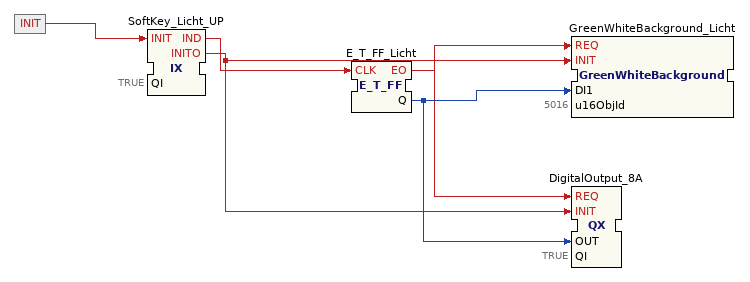
      FBS
        E_T_FF_Licht : E_T_FF;
        GreenWhiteBackground_Licht : GreenWhiteBackground(u16ObjId := 5016);
        DigitalOutput_8A : QX(QI := TRUE);
        SoftKey_Licht_UP : IX(QI := TRUE);
      END_FBS
      EVENT_CONNECTIONS
        SoftKey_Licht_UP.IND TO E_T_FF_Licht.CLK;
        E_T_FF_Licht.EO TO DigitalOutput_8A.REQ;
        E_T_FF_Licht.EO TO GreenWhiteBackground_Licht.REQ;
        SoftKey_Licht_UP.INITO TO GreenWhiteBackground_Licht.INIT;
        SoftKey_Licht_UP.INITO TO DigitalOutput_8A.INIT;
        INIT TO SoftKey_Licht_UP.INIT;
      END_CONNECTIONS
      DATA_CONNECTIONS
        E_T_FF_Licht.Q TO DigitalOutput_8A.OUT;
        E_T_FF_Licht.Q TO GreenWhiteBackground_Licht.DI1;
      END_CONNECTIONS
    END_SUBAPPLICATION
  END_APPLICATION
  APPLICATION Abscheider
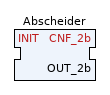
    SUBAPPLICATION Abscheider (* Abscheider *)
      EVENT_INPUT
        INIT; (* Service Initialization *)
      END_EVENT
      EVENT_OUTPUT
        CNF_2b; (* Execution Confirmation *)
      END_EVENT
      VAR_OUTPUT
        OUT_2b : BOOL;
      END_VAR
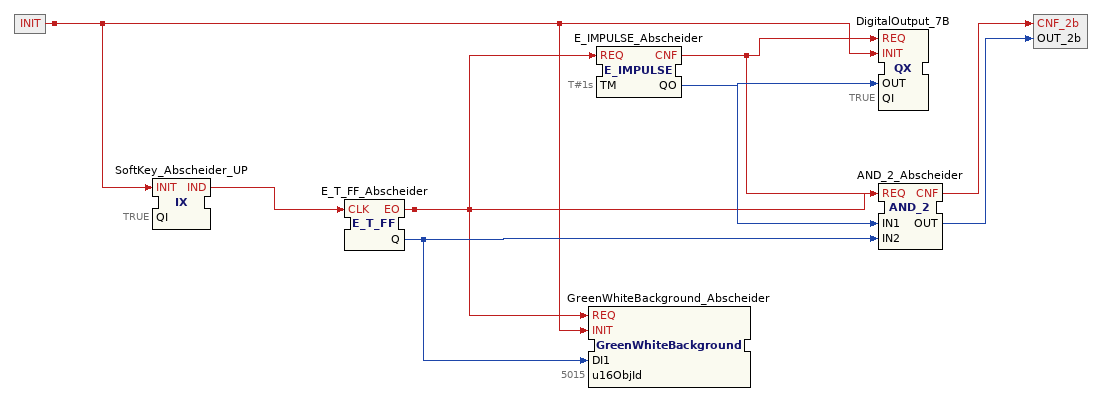
      FBS
        SoftKey_Abscheider_UP : IX(QI := TRUE);
        E_IMPULSE_Abscheider : E_IMPULSE(TM := T#1s);
        E_T_FF_Abscheider : E_T_FF;
        DigitalOutput_7B : QX(QI := TRUE);
        AND_2_Abscheider : AND_2;
        GreenWhiteBackground_Abscheider : GreenWhiteBackground(u16ObjId := 5015);
      END_FBS
      EVENT_CONNECTIONS
        SoftKey_Abscheider_UP.IND TO E_T_FF_Abscheider.CLK;
        E_T_FF_Abscheider.EO TO E_IMPULSE_Abscheider.REQ;
        E_IMPULSE_Abscheider.CNF TO AND_2_Abscheider.REQ;
        E_IMPULSE_Abscheider.CNF TO DigitalOutput_7B.REQ;
        E_T_FF_Abscheider.EO TO AND_2_Abscheider.REQ;
        E_T_FF_Abscheider.EO TO GreenWhiteBackground_Abscheider.REQ;
        INIT TO SoftKey_Abscheider_UP.INIT;
        AND_2_Abscheider.CNF TO CNF_2b;
        INIT TO GreenWhiteBackground_Abscheider.INIT;
        INIT TO DigitalOutput_7B.INIT;
      END_CONNECTIONS
      DATA_CONNECTIONS
        E_IMPULSE_Abscheider.QO TO AND_2_Abscheider.IN1;
        E_IMPULSE_Abscheider.QO TO DigitalOutput_7B.OUT;
        E_T_FF_Abscheider.Q TO AND_2_Abscheider.IN2;
        E_T_FF_Abscheider.Q TO GreenWhiteBackground_Abscheider.DI1;
        AND_2_Abscheider.OUT TO OUT_2b;
      END_CONNECTIONS
    END_SUBAPPLICATION
  END_APPLICATION
  APPLICATION Automatik
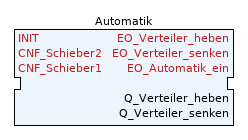
    SUBAPPLICATION Automatik (* Automatik *)
      EVENT_INPUT
        INIT;
        CNF_Schieber2;
        CNF_Schieber1;
      END_EVENT
      EVENT_OUTPUT
        EO_Verteiler_heben;
        EO_Verteiler_senken;
        EO_Automatik_ein;
      END_EVENT
      VAR_OUTPUT
        Q_Verteiler_heben : BOOL;
        Q_Verteiler_senken : BOOL;
      END_VAR
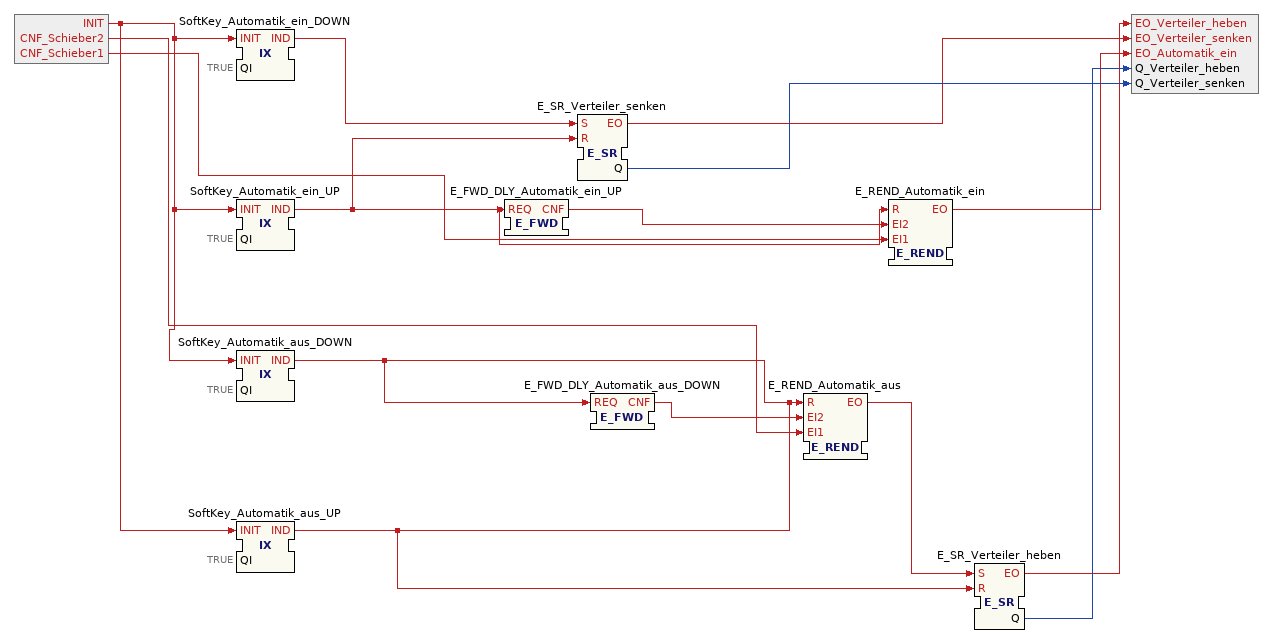
      FBS
        SoftKey_Automatik_aus_DOWN : IX(QI := TRUE);
        E_SR_Verteiler_heben : E_SR;
        E_FWD_DLY_Automatik_aus_DOWN : E_FWD;
        SoftKey_Automatik_ein_DOWN : IX(QI := TRUE);
        SoftKey_Automatik_ein_UP : IX(QI := TRUE);
        SoftKey_Automatik_aus_UP : IX(QI := TRUE);
        E_REND_Automatik_aus : E_REND;
        E_FWD_DLY_Automatik_ein_UP : E_FWD;
        E_SR_Verteiler_senken : E_SR;
        E_REND_Automatik_ein : E_REND;
      END_FBS
      EVENT_CONNECTIONS
        SoftKey_Automatik_aus_DOWN.IND TO E_FWD_DLY_Automatik_aus_DOWN.REQ;
        SoftKey_Automatik_aus_DOWN.IND TO E_REND_Automatik_aus.R;
        E_REND_Automatik_aus.EO TO E_SR_Verteiler_heben.S;
        SoftKey_Automatik_aus_UP.IND TO E_SR_Verteiler_heben.R;
        E_FWD_DLY_Automatik_aus_DOWN.CNF TO E_REND_Automatik_aus.EI2;
        SoftKey_Automatik_ein_DOWN.IND TO E_SR_Verteiler_senken.S;
        SoftKey_Automatik_ein_UP.IND TO E_SR_Verteiler_senken.R;
        SoftKey_Automatik_ein_UP.IND TO E_FWD_DLY_Automatik_ein_UP.REQ;
        SoftKey_Automatik_ein_UP.IND TO E_REND_Automatik_ein.R;
        SoftKey_Automatik_aus_UP.IND TO E_REND_Automatik_aus.R;
        E_FWD_DLY_Automatik_ein_UP.CNF TO E_REND_Automatik_ein.EI2;
        INIT TO SoftKey_Automatik_aus_DOWN.INIT;
        E_SR_Verteiler_heben.EO TO EO_Verteiler_heben;
        INIT TO SoftKey_Automatik_ein_DOWN.INIT;
        INIT TO SoftKey_Automatik_ein_UP.INIT;
        INIT TO SoftKey_Automatik_aus_UP.INIT;
        CNF_Schieber2 TO E_REND_Automatik_aus.EI1;
        E_SR_Verteiler_senken.EO TO EO_Verteiler_senken;
        CNF_Schieber1 TO E_REND_Automatik_ein.EI1;
        E_REND_Automatik_ein.EO TO EO_Automatik_ein;
      END_CONNECTIONS
      DATA_CONNECTIONS
        E_SR_Verteiler_heben.Q TO Q_Verteiler_heben;
        E_SR_Verteiler_senken.Q TO Q_Verteiler_senken;
      END_CONNECTIONS
    END_SUBAPPLICATION
  END_APPLICATION
  APPLICATION Vorsteuerventil_2B
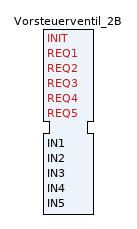
    SUBAPPLICATION Vorsteuerventil_2B (* Vorsteuerventil_2B *)
      EVENT_INPUT
        INIT;
        REQ1;
        REQ2;
        REQ3;
        REQ4;
        REQ5;
      END_EVENT
      VAR_INPUT
        IN1 : BOOL;
        IN2 : BOOL;
        IN3 : BOOL;
        IN4 : BOOL;
        IN5 : BOOL;
      END_VAR
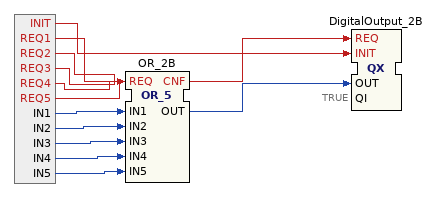
      FBS
        DigitalOutput_2B : QX(QI := TRUE);
        OR_2B : OR_5;
      END_FBS
      EVENT_CONNECTIONS
        OR_2B.CNF TO DigitalOutput_2B.REQ;
        INIT TO DigitalOutput_2B.INIT;
        REQ1 TO OR_2B.REQ;
        REQ2 TO OR_2B.REQ;
        REQ3 TO OR_2B.REQ;
        REQ4 TO OR_2B.REQ;
        REQ5 TO OR_2B.REQ;
      END_CONNECTIONS
      DATA_CONNECTIONS
        OR_2B.OUT TO DigitalOutput_2B.OUT;
        IN1 TO OR_2B.IN1;
        IN2 TO OR_2B.IN2;
        IN3 TO OR_2B.IN3;
        IN4 TO OR_2B.IN4;
        IN5 TO OR_2B.IN5;
      END_CONNECTIONS
    END_SUBAPPLICATION
  END_APPLICATION
  DEVICE FORTE_PC : FORTE_PC(MGR_ID := "192.168.4.1:61499")
    {SET_ATTRIBUTE(Profile, DynamicTypeLoad)}
    {SET_ATTRIBUTE(FBType, GEN_E_MUX, F_LT, E_CTD, E_STOPWATCH, F_LIMIT, UT_AuxiliaryInputMapping, UT_ButtonMapping_UP, F_TIME_IN_S_TO_UDINT, F_TAN, COLOR_BLACK, F_ACOS, QD, COLOR_WHITE, COLOR_OLIVE, E_MERGE, DataPanel_xDB0808_DIO_SAE_J1939, EMB_RES, COLOR_CYAN, ID, E_DEMUX, GEN_SUBL, QW, QX, F_MUL, IW, IX, Q_ChangePolygonScale, F_LE, GEN_SUBSCRIBE, F_ATAN, GEN_AND, F_SIN, F_LN, GEN_CLIENT, F_NOT, COLOR_MAROON, GEN_SERVER, GEN_PUBL, Q_SelectActiveWorkingSet, E_IMPULSE, RMT_RES, COLOR_RED, UT_ButtonMapping_HOLD, GEN_OR, E_D_FF, E_CYCLE, UT_ButtonMapping, E_R_TRIG, COLOR_TEAL, COLOR_BLUE, Q_ActiveMask, F_GE, E_F_TRIG, GreenWhiteBackground, E_RS, F_MUX_2, DEV_MGR, E_SPLIT, E_FWD, E_CTUD, UT_SoftkeyMapping_UP, F_EQ, E_T_FF, E_RDELAY, UT_ButtonMapping_DOWN, F_MOD, E_RTimeOut, F_NE, CbVtStatus, Q_ObjEnableDisable, F_TIME_IN_NS_TO_UDINT, FB_RANDOM, F_EXP, E_SELECT, GEN_PUBLISH, F_TIME_IN_MS_TO_UDINT, E_CTUD_UDINT, Q_CtrlAudioSignal, E_TRAIN, OUT_ANY_CONSOLE, F_SUB, Q_ChangeObjectLabel, F_GT, COLOR_YELLOW, GEN_E_DEMUX, F_LOG, F_SQRT, DataPanel_xDB_16_DO_SAE_J1939, E_SR, COLOR_NAVY, GEN_XOR, Q_ChildLocation, F_MIN, E_SWITCH, E_RESTART, E_PERMIT, UT_SoftkeyMapping_HOLD, F_SEL, Q_ChangePolygonPoint, UT_SoftkeyMapping, F_MAX, E_TimeOut, COLOR_SILVER, Q_BackgroundColour, COLOR_MAGENTA, UT_SoftkeyMapping_DOWN, Q_Attribute, COLOR_LIME, COLOR_GREEN, COLOR_GREY, COLOR_PURPLE, F_ABS, E_DELAY, GEN_ADD, F_COS, Q_ObjHideShow, Q_StringValue, F_TIME_IN_US_TO_UDINT, E_CTU, Q_NumericValue, Q_ChildPosition, E_REND, F_ASIN, F_DIV)} (* created during deployment *)
    RESOURCE EMB_RES : EMB_RES
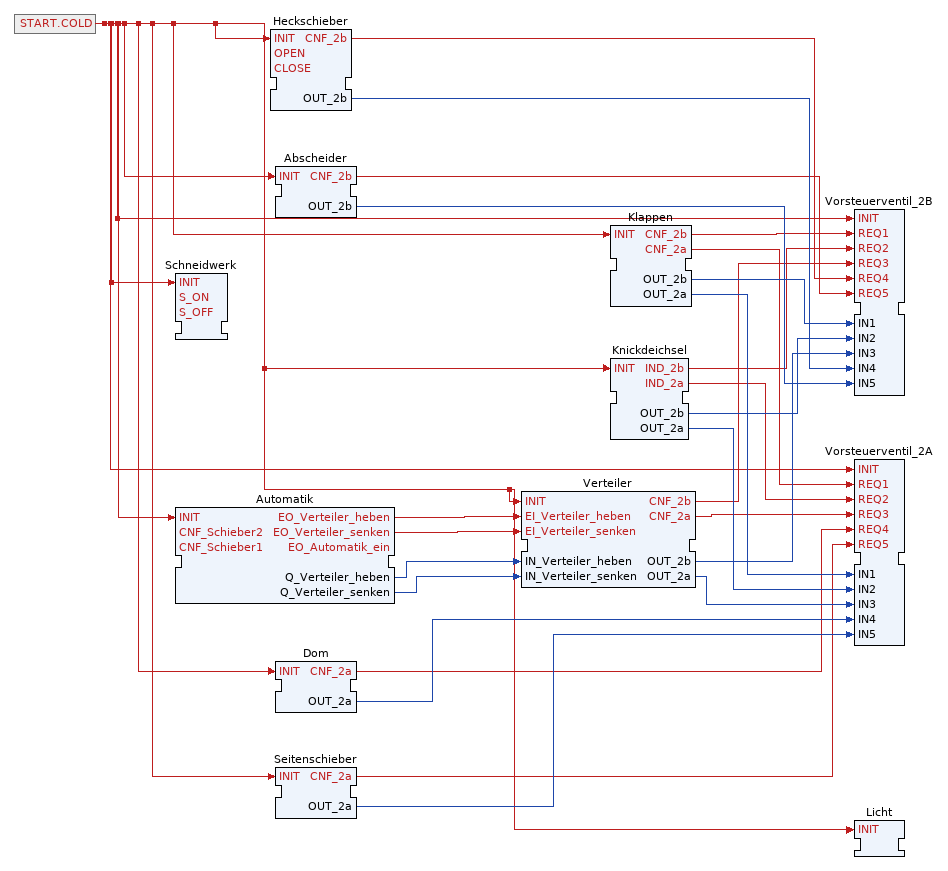
      SUBAPPLICATION Vorsteuerventil_2A
        EVENT_INPUT
          INIT;
          REQ1;
          REQ2;
          REQ3;
          REQ4;
          REQ5;
        END_EVENT
        VAR_INPUT
          IN1 : BOOL;
          IN2 : BOOL;
          IN3 : BOOL;
          IN4 : BOOL;
          IN5 : BOOL;
        END_VAR
      END_SUBAPPLICATION
      SUBAPPLICATION Vorsteuerventil_2B
        EVENT_INPUT
          INIT;
          REQ1;
          REQ2;
          REQ3;
          REQ4;
          REQ5;
        END_EVENT
        VAR_INPUT
          IN1 : BOOL;
          IN2 : BOOL;
          IN3 : BOOL;
          IN4 : BOOL;
          IN5 : BOOL;
        END_VAR
      END_SUBAPPLICATION
      SUBAPPLICATION Abscheider
        EVENT_INPUT
          INIT; (* Service Initialization *)
        END_EVENT
        EVENT_OUTPUT
          CNF_2b; (* Execution Confirmation *)
        END_EVENT
        VAR_OUTPUT
          OUT_2b : BOOL;
        END_VAR
      END_SUBAPPLICATION
      SUBAPPLICATION Dom
        EVENT_INPUT
          INIT;
        END_EVENT
        EVENT_OUTPUT
          CNF_2a;
        END_EVENT
        VAR_OUTPUT
          OUT_2a : BOOL;
        END_VAR
      END_SUBAPPLICATION
      SUBAPPLICATION Seitenschieber
        EVENT_INPUT
          INIT;
        END_EVENT
        EVENT_OUTPUT
          CNF_2a;
        END_EVENT
        VAR_OUTPUT
          OUT_2a : BOOL;
        END_VAR
      END_SUBAPPLICATION
      SUBAPPLICATION Heckschieber
        EVENT_INPUT
          INIT;
          OPEN;
          CLOSE;
        END_EVENT
        EVENT_OUTPUT
          CNF_2b;
        END_EVENT
        VAR_OUTPUT
          OUT_2b : BOOL;
        END_VAR
      END_SUBAPPLICATION
      SUBAPPLICATION Klappen
        EVENT_INPUT
          INIT;
        END_EVENT
        EVENT_OUTPUT
          CNF_2b;
          CNF_2a;
        END_EVENT
        VAR_OUTPUT
          OUT_2b : BOOL;
          OUT_2a : BOOL;
        END_VAR
      END_SUBAPPLICATION
      SUBAPPLICATION Knickdeichsel
        EVENT_INPUT
          INIT;
        END_EVENT
        EVENT_OUTPUT
          IND_2b;
          IND_2a;
        END_EVENT
        VAR_OUTPUT
          OUT_2b : BOOL;
          OUT_2a : BOOL;
        END_VAR
      END_SUBAPPLICATION
      SUBAPPLICATION Licht
        EVENT_INPUT
          INIT; (* Service Initialization *)
        END_EVENT
      END_SUBAPPLICATION
      SUBAPPLICATION Schneidwerk
        EVENT_INPUT
          INIT;
          S_ON;
          S_OFF;
        END_EVENT
      END_SUBAPPLICATION
      SUBAPPLICATION Automatik
        EVENT_INPUT
          INIT;
          CNF_Schieber2;
          CNF_Schieber1;
        END_EVENT
        EVENT_OUTPUT
          EO_Verteiler_heben;
          EO_Verteiler_senken;
          EO_Automatik_ein;
        END_EVENT
        VAR_OUTPUT
          Q_Verteiler_heben : BOOL;
          Q_Verteiler_senken : BOOL;
        END_VAR
      END_SUBAPPLICATION
      SUBAPPLICATION Verteiler
        EVENT_INPUT
          INIT;
          EI_Verteiler_heben;
          EI_Verteiler_senken;
        END_EVENT
        EVENT_OUTPUT
          CNF_2b;
          CNF_2a;
        END_EVENT
        VAR_INPUT
          IN_Verteiler_heben : BOOL;
          IN_Verteiler_senken : BOOL;
        END_VAR
        VAR_OUTPUT
          OUT_2b : BOOL;
          OUT_2a : BOOL;
        END_VAR
      END_SUBAPPLICATION
      EVENT_CONNECTIONS
        START.COLD TO Vorsteuerventil_2A.INIT;
        START.COLD TO Vorsteuerventil_2B.INIT;
        START.COLD TO Abscheider.INIT;
        Abscheider.CNF_2b TO Vorsteuerventil_2B.REQ5;
        START.COLD TO Dom.INIT;
        Dom.CNF_2a TO Vorsteuerventil_2A.REQ4;
        START.COLD TO Seitenschieber.INIT;
        Seitenschieber.CNF_2a TO Vorsteuerventil_2A.REQ5;
        Heckschieber.CNF_2b TO Vorsteuerventil_2B.REQ4;
        START.COLD TO Klappen.INIT;
        Klappen.CNF_2b TO Vorsteuerventil_2B.REQ1;
        Klappen.CNF_2a TO Vorsteuerventil_2A.REQ1;
        START.COLD TO Knickdeichsel.INIT;
        Knickdeichsel.IND_2b TO Vorsteuerventil_2B.REQ2;
        Knickdeichsel.IND_2a TO Vorsteuerventil_2A.REQ2;
        START.COLD TO Heckschieber.INIT;
        START.COLD TO Licht.INIT;
        START.COLD TO Schneidwerk.INIT;
        START.COLD TO Automatik.INIT;
        Verteiler.CNF_2b TO Vorsteuerventil_2B.REQ3;
        Verteiler.CNF_2a TO Vorsteuerventil_2A.REQ3;
        START.COLD TO Verteiler.INIT;
        Automatik.EO_Verteiler_senken TO Verteiler.EI_Verteiler_senken;
        Automatik.EO_Verteiler_heben TO Verteiler.EI_Verteiler_heben;
      END_CONNECTIONS
      DATA_CONNECTIONS
        Abscheider.OUT_2b TO Vorsteuerventil_2B.IN5;
        Dom.OUT_2a TO Vorsteuerventil_2A.IN4;
        Seitenschieber.OUT_2a TO Vorsteuerventil_2A.IN5;
        Heckschieber.OUT_2b TO Vorsteuerventil_2B.IN4;
        Klappen.OUT_2b TO Vorsteuerventil_2B.IN1;
        Klappen.OUT_2a TO Vorsteuerventil_2A.IN1;
        Knickdeichsel.OUT_2b TO Vorsteuerventil_2B.IN2;
        Knickdeichsel.OUT_2a TO Vorsteuerventil_2A.IN2;
        Automatik.Q_Verteiler_heben TO Verteiler.IN_Verteiler_heben;
        Automatik.Q_Verteiler_senken TO Verteiler.IN_Verteiler_senken;
        Verteiler.OUT_2a TO Vorsteuerventil_2A.IN3;
        Verteiler.OUT_2b TO Vorsteuerventil_2B.IN3;
      END_CONNECTIONS
    END_RESOURCE
  END_DEVICE
  MAPPINGS
    Vorsteuerventil_2A.Vorsteuerventil_2A ON FORTE_PC.EMB_RES.Vorsteuerventil_2A;
    Vorsteuerventil_2B.Vorsteuerventil_2B ON FORTE_PC.EMB_RES.Vorsteuerventil_2B;
    Abscheider.Abscheider ON FORTE_PC.EMB_RES.Abscheider;
    Dom.Dom ON FORTE_PC.EMB_RES.Dom;
    Seitenschieber.Seitenschieber ON FORTE_PC.EMB_RES.Seitenschieber;
    Heckschieber.Heckschieber ON FORTE_PC.EMB_RES.Heckschieber;
    Klappen.Klappen ON FORTE_PC.EMB_RES.Klappen;
    Knickdeichsel.Knickdeichsel ON FORTE_PC.EMB_RES.Knickdeichsel;
    Licht.Licht ON FORTE_PC.EMB_RES.Licht;
    Schneidwerk.Schneidwerk ON FORTE_PC.EMB_RES.Schneidwerk;
    Automatik.Automatik ON FORTE_PC.EMB_RES.Automatik;
    Verteiler.Verteiler ON FORTE_PC.EMB_RES.Verteiler;
  END_MAPPINGS
  SEGMENTS
    Ethernet : Ethernet;
  END_SEGMENTS
  LINKS
    FORTE_PC => Ethernet;
  END_LINKS
END_SYSTEM
